INTERFACE I_CalculateThickness


METHOD PUBLIC Calculate
VAR_INPUT
    fDesiredTransmission : LREAL; // [1]
    fPhotonEnergy : LREAL; // [eV]
END_VAR
VAR_OUTPUT
    fThickness : LREAL; // [mm]
END_VAR
END_METHOD

END_INTERFACE

(* stored: Version 1.1.0.1
   Itf I_CalculateThickness: Id {7ca46989-50f7-43cc-9cc6-210fcb015be6}
   Method Calculate: Id {11c99484-72d2-4339-937d-7b0d2d2530db} *)
